(**************************************************************************************
CopyRight Atlantis Operations UK Ltd 2015
AR500 TCS

Function Block Purpose:
Need to ensure that we have access rights controls being verified here 
even though this is also controlled by the SCADA. The Safety can also be
managed through this function block. Use the TwinCAT user level controls
to this end.

Version history: Created with TwinCat V 2.11.2248
04/08/15	V 0.01		NSM - ODT First Draft
***************************************************************************************)

FUNCTION_BLOCK FB_AlarmResetAccessCtrl
VAR_INPUT
END_VAR
VAR_OUTPUT
END_VAR
VAR
	bDummy: BOOL;
END_VAR

bDummy:=FALSE;

END_FUNCTION_BLOCK

(* stored: Version 1.1.0.1, ProductVersion 3.1.4024.11
   POU FB_AlarmResetAccessCtrl: Id {90d359b3-5ce6-4319-a8cb-ff7e024ae2ae}, SpecialFunc None *)
